/// This struct contains variables that
/// * are read from outside (e.g. HMI) to retrieve information about the unit's current state and (temporary) parameters (= `publish`) 
/// * are written from outside (e.g. HMI) to control the unit via ADS (= `subscribe`) 
TYPE DrillingCom :
STRUCT
  Publish : DrillingComPublish;
  Subscribe : DrillingComSubscribe;
END_STRUCT
END_TYPE

(* stored: Version 1.1.0.1
   DUT DrillingCom: Id {1a1e29aa-0a29-4d6a-b391-6397aff2d231} *)
